# EPICS autosave request: ADApp/Db/NDColorConvert_settings.req
$(P)$(R)ColorModeOut
